{attribute 'GeneratedUsingTerminal: EP9224-1037-0017'}
{attribute addProperty BoxType "EP9224-1037-0017"}
{attribute addProperty Id "InfoDataAT %I*InfoData_6F19DB2B2"}
{attribute addProperty CRC "532711307"}
{attribute addProperty Size "2"}
TYPE EP9224_1FC0878B EXTENDS EtcSlaveTerminalBase_947E5A46 :
STRUCT
	{attribute addProperty Name "InfoData"}
	InfoData : InfoData_6F19DB2B;
END_STRUCT
END_TYPE

(* stored: Version 1.2.0.0, ProductVersion 3.1.4024.9
   DUT EP9224_1FC0878B: Id {23a2b830-2933-402a-b9dd-0b11930ed7e4} *)
